// TIA Portal V21 export
DATA_BLOCK "SegnaliMacchina"   // DB27
{ S7_Optimized_Access := 'TRUE' }
// stored: MemoryReserve 0
   VAR RETAIN
      S : Array[0.."K_NumSegnaleMacchina"] of "Std_SegnaliMacchina";
   END_VAR
BEGIN
   // S[1] : QCI
   // S[2] : CFT
   // S[1].SR[0].Digitali[1] : ChiamataProdotto
   // S[2].SR[0].Digitali[1] : ImpiantoInSterilizzazione
   // S[2].SR[0].Digitali[2] : ImpiantoInLavaggio
   // S[2].SR[0].Digitali[3] : ImpulsiPompaPistoni
   // S[2].SR[0].Digitali[4] : ImpiantoInProduzione
   // S[2].SR[0].Digitali[5] : ProdottoDisponibile
   S[0].SR[0].Digitali[0..31].In.Segnale := FALSE;
   S[0].SR[1].Digitali[0..31].In.Segnale := FALSE;
   S[1].SR[0].Digitali[0..31].In.Segnale := FALSE;
   S[1].SR[1].Digitali[0..31].In.Segnale := FALSE;
   S[2].SR[0].Digitali[0..31].In.Segnale := FALSE;
   S[2].SR[1].Digitali[0..31].In.Segnale := FALSE;
   S[0].SR[0].Digitali[0..31].Prm.AbilitaScadenzaForzatura := FALSE;
   S[0].SR[1].Digitali[0..31].Prm.AbilitaScadenzaForzatura := FALSE;
   S[1].SR[0].Digitali[0..31].Prm.AbilitaScadenzaForzatura := FALSE;
   S[1].SR[1].Digitali[0..31].Prm.AbilitaScadenzaForzatura := FALSE;
   S[2].SR[0].Digitali[0].Prm.AbilitaScadenzaForzatura := FALSE;
   S[2].SR[0].Digitali[1..5].Prm.AbilitaScadenzaForzatura := TRUE;
   S[2].SR[0].Digitali[6..31].Prm.AbilitaScadenzaForzatura := FALSE;
   S[2].SR[1].Digitali[0].Prm.AbilitaScadenzaForzatura := FALSE;
   S[2].SR[1].Digitali[1].Prm.AbilitaScadenzaForzatura := TRUE;
   S[2].SR[1].Digitali[2..31].Prm.AbilitaScadenzaForzatura := FALSE;
   S[0].SR[0].Digitali[0..31].Prm.TempoScadenzaForzatura.IN := FALSE;
   S[0].SR[1].Digitali[0..31].Prm.TempoScadenzaForzatura.IN := FALSE;
   S[1].SR[0].Digitali[0..31].Prm.TempoScadenzaForzatura.IN := FALSE;
   S[1].SR[1].Digitali[0..31].Prm.TempoScadenzaForzatura.IN := FALSE;
   S[2].SR[0].Digitali[0..31].Prm.TempoScadenzaForzatura.IN := FALSE;
   S[2].SR[1].Digitali[0..31].Prm.TempoScadenzaForzatura.IN := FALSE;
   S[0].SR[0].Digitali[0..31].Prm.TempoScadenzaForzatura.O := FALSE;
   S[0].SR[1].Digitali[0..31].Prm.TempoScadenzaForzatura.O := FALSE;
   S[1].SR[0].Digitali[0..31].Prm.TempoScadenzaForzatura.O := FALSE;
   S[1].SR[1].Digitali[0..31].Prm.TempoScadenzaForzatura.O := FALSE;
   S[2].SR[0].Digitali[0..31].Prm.TempoScadenzaForzatura.O := FALSE;
   S[2].SR[1].Digitali[0..31].Prm.TempoScadenzaForzatura.O := FALSE;
   S[0].SR[0].Digitali[0..31].Prm.TempoScadenzaForzatura.Preset := 0.0;
   S[0].SR[1].Digitali[0..31].Prm.TempoScadenzaForzatura.Preset := 0.0;
   S[1].SR[0].Digitali[0].Prm.TempoScadenzaForzatura.Preset := 0.0;
   S[1].SR[0].Digitali[1].Prm.TempoScadenzaForzatura.Preset := 300.0;
   S[1].SR[0].Digitali[2..31].Prm.TempoScadenzaForzatura.Preset := 0.0;
   S[1].SR[1].Digitali[0..31].Prm.TempoScadenzaForzatura.Preset := 0.0;
   S[2].SR[0].Digitali[0].Prm.TempoScadenzaForzatura.Preset := 0.0;
   S[2].SR[0].Digitali[1..5].Prm.TempoScadenzaForzatura.Preset := 300.0;
   S[2].SR[0].Digitali[6..31].Prm.TempoScadenzaForzatura.Preset := 0.0;
   S[2].SR[1].Digitali[0].Prm.TempoScadenzaForzatura.Preset := 0.0;
   S[2].SR[1].Digitali[1].Prm.TempoScadenzaForzatura.Preset := 300.0;
   S[2].SR[1].Digitali[2..31].Prm.TempoScadenzaForzatura.Preset := 0.0;
   S[0].SR[0].Digitali[0..31].Prm.TempoScadenzaForzatura.TempoTrascorso := 0.0;
   S[0].SR[1].Digitali[0..31].Prm.TempoScadenzaForzatura.TempoTrascorso := 0.0;
   S[1].SR[0].Digitali[0..31].Prm.TempoScadenzaForzatura.TempoTrascorso := 0.0;
   S[1].SR[1].Digitali[0..31].Prm.TempoScadenzaForzatura.TempoTrascorso := 0.0;
   S[2].SR[0].Digitali[0..31].Prm.TempoScadenzaForzatura.TempoTrascorso := 0.0;
   S[2].SR[1].Digitali[0..31].Prm.TempoScadenzaForzatura.TempoTrascorso := 0.0;
   S[0].SR[0].Digitali[0..31].Hmi.ForzaturaOn := FALSE;
   S[0].SR[1].Digitali[0..31].Hmi.ForzaturaOn := FALSE;
   S[1].SR[0].Digitali[0..31].Hmi.ForzaturaOn := FALSE;
   S[1].SR[1].Digitali[0..31].Hmi.ForzaturaOn := FALSE;
   S[2].SR[0].Digitali[0..31].Hmi.ForzaturaOn := FALSE;
   S[2].SR[1].Digitali[0..31].Hmi.ForzaturaOn := FALSE;
   S[0].SR[0].Digitali[0..31].Hmi.ForzaturaOff := FALSE;
   S[0].SR[1].Digitali[0..31].Hmi.ForzaturaOff := FALSE;
   S[1].SR[0].Digitali[0..31].Hmi.ForzaturaOff := FALSE;
   S[1].SR[1].Digitali[0..31].Hmi.ForzaturaOff := FALSE;
   S[2].SR[0].Digitali[0..31].Hmi.ForzaturaOff := FALSE;
   S[2].SR[1].Digitali[0..31].Hmi.ForzaturaOff := FALSE;
   S[0].SR[0].Digitali[0..31].Hmi.Stato := 0;
   S[0].SR[1].Digitali[0..31].Hmi.Stato := 0;
   S[1].SR[0].Digitali[0].Hmi.Stato := 0;
   S[1].SR[0].Digitali[1].Hmi.Stato := 1;
   S[1].SR[0].Digitali[2..31].Hmi.Stato := 0;
   S[1].SR[1].Digitali[0..31].Hmi.Stato := 0;
   S[2].SR[0].Digitali[0..3].Hmi.Stato := 0;
   S[2].SR[0].Digitali[4..5].Hmi.Stato := 1;
   S[2].SR[0].Digitali[6..31].Hmi.Stato := 0;
   S[2].SR[1].Digitali[0].Hmi.Stato := 0;
   S[2].SR[1].Digitali[1].Hmi.Stato := 1;
   S[2].SR[1].Digitali[2..3].Hmi.Stato := 0;
   S[2].SR[1].Digitali[4..5].Hmi.Stato := 1;
   S[2].SR[1].Digitali[6..31].Hmi.Stato := 0;
   S[0].SR[0].Digitali[0..31].Out.Segnale := FALSE;
   S[0].SR[1].Digitali[0..31].Out.Segnale := FALSE;
   S[1].SR[0].Digitali[0].Out.Segnale := FALSE;
   S[1].SR[0].Digitali[1].Out.Segnale := TRUE;
   S[1].SR[0].Digitali[2..31].Out.Segnale := FALSE;
   S[1].SR[1].Digitali[0..31].Out.Segnale := FALSE;
   S[2].SR[0].Digitali[0..3].Out.Segnale := FALSE;
   S[2].SR[0].Digitali[4..5].Out.Segnale := TRUE;
   S[2].SR[0].Digitali[6..31].Out.Segnale := FALSE;
   S[2].SR[1].Digitali[0].Out.Segnale := FALSE;
   S[2].SR[1].Digitali[1].Out.Segnale := TRUE;
   S[2].SR[1].Digitali[2..3].Out.Segnale := FALSE;
   S[2].SR[1].Digitali[4..5].Out.Segnale := TRUE;
   S[2].SR[1].Digitali[6..31].Out.Segnale := FALSE;
   S[0].SR[0]."DInt"[0..19] := 0;
   S[0].SR[1]."DInt"[0..19] := 0;
   S[1].SR[0]."DInt"[0..19] := 0;
   S[1].SR[1]."DInt"[0..19] := 0;
   S[2].SR[0]."DInt"[0..19] := 0;
   S[2].SR[1]."DInt"[0..19] := 0;
   S[0].SR[0]."Real"[0..19] := 0.0;
   S[0].SR[1]."Real"[0..19] := 0.0;
   S[1].SR[0]."Real"[0..19] := 0.0;
   S[1].SR[1]."Real"[0..19] := 0.0;
   S[2].SR[0]."Real"[0..19] := 0.0;
   S[2].SR[1]."Real"[0..19] := 0.0;
   S[0].SR[0..1].Prm.Abilitazione := FALSE;
   S[1].SR[0..1].Prm.Abilitazione := FALSE;
   S[2].SR[0..1].Prm.Abilitazione := FALSE;
   S[0..2].Prm.Watchdog.Bit.Abilitato := FALSE;
   S[0..2].Prm.Watchdog.Bit.RestituisciWatchdog := FALSE;
   S[0..2].Prm.Watchdog.Bit.RestituisciNegato := FALSE;
   S[0..2].Prm.Watchdog.Incrementale.Abilitato := FALSE;
   S[0].Prm.TipoComunicazione := 0;
   S[1].Prm.TipoComunicazione := 1;
   S[2].Prm.TipoComunicazione := 0;
   S[0].Allarmi."A"[0..3].Abilitato := FALSE;
   S[1].Allarmi."A"[0..3].Abilitato := FALSE;
   S[2].Allarmi."A"[0..3].Abilitato := FALSE;
   S[0].Allarmi."A"[0..3].Stato := FALSE;
   S[1].Allarmi."A"[0..3].Stato := FALSE;
   S[2].Allarmi."A"[0..3].Stato := FALSE;
   S[0].Allarmi."A"[0..3].Silenziato := FALSE;
   S[1].Allarmi."A"[0..3].Silenziato := FALSE;
   S[2].Allarmi."A"[0..3].Silenziato := FALSE;
   S[0].Allarmi."A"[0].EnWarnHmi := FALSE;
   S[0].Allarmi."A"[1..3].EnWarnHmi := TRUE;
   S[1].Allarmi."A"[0].EnWarnHmi := FALSE;
   S[1].Allarmi."A"[1..3].EnWarnHmi := TRUE;
   S[2].Allarmi."A"[0].EnWarnHmi := FALSE;
   S[2].Allarmi."A"[1..3].EnWarnHmi := TRUE;
   S[0].Allarmi."A"[0..3].EnCadutaCiclo := FALSE;
   S[1].Allarmi."A"[0..3].EnCadutaCiclo := FALSE;
   S[2].Allarmi."A"[0..3].EnCadutaCiclo := FALSE;
   S[0..2].Allarmi.WordHmi := 16#0000;
END_DATA_BLOCK
